// TIA Portal V20 export
DATA_BLOCK "BK06"   // DB201
// stored: MemoryReserve 100
   VAR
      "X10-1 NG & MANUAL INPUT CYLINDER UP" : Bool;
      "X11-1 MAGAZINE LOCK CYLINDER DOWN" : Bool;
      "X12-1 NG & MANUAL INPUT PAD VACUUM PRESSURE SWITCH" : Bool;
      "X13-1 NG & MANUAL INPUT LIMIT SENSOR(-)" : Bool;
      "X14-1 NG & MANUAL INPUT LIMIT SENSOR(+)" : Bool;
      "X15-1 NG & MANUAL INPUT MAGAZINE LIMIT SENSOR(-)" : Bool;
      "X16-1 NG & MANUAL INPUT MAGAZINE LIMIT SENSOR(+)" : Bool;
      "X17-1 NG & MANUAL INPUT MAGAZINE ELECTRODE DETECTION SENSOR" : Bool;
      "X10-2 NG & MANUAL INPUT CYLINDER DOWN" : Bool;
      "X11-2 MAGAZINE LOCK CYLINDER UP" : Bool;
      "X12-2 NG & MANUAL INPUT VIBRATOR VACUUM PRESSURE SWITCH" : Bool;
      "X13-2 NG & MANUAL INPUT HOMING SENSOR" : Bool;
      "X14-2 NG & MANUAL INPUT ELECTRODE DETECTION SENSOR" : Bool;
      "X15-2 NG & MANUAL INPUT MAGAZINE HOMING SENSOR" : Bool;
      "X16-2 SPARE" : Bool;
      "X17-2 NG & MANUAL INPUT MAGAZINE DETECTION SENSOR" : Bool;
   END_VAR
BEGIN
END_DATA_BLOCK
